PROGRAM MAIN
VAR
  // ── Core robot interface (library FBs) ────────────────────────────────────
  fbStatus     : FB_FanucStatus;        // DI0 byte array → stStatus struct
  fbControl    : FB_FanucControl;       // stControl struct → DO0 byte array
  fbEnable     : FB_FanucEnable;        // Enable sequence state machine
  fbFaultReset : FB_FanucFaultReset;    // Fault reset pulse – FAULT_RESET (UI[5])
  fbStart      : FB_FanucStartProgram;  // Program start (RSR / PNS)
  fbCycleStop  : FB_FanucCycleStop;     // Cycle Stop – CSTOPI (UI[4])
  fbHoming     : FB_FanucHoming;        // Homing sequence – HOME (UI[7])
  stStatus     : ST_FanucStatus;        // Live robot status (inputs)
  stControl    : ST_FanucControl;       // Combined control command (outputs)

  // ── Enable command ────────────────────────────────────────────────────────
  bEnableRobot : BOOL;               // Set TRUE to start enable sequence

  // ── External interlock signals (wire from application safety logic / HMI) ─
  bExtIMSTP  : BOOL;  // Normally Closed: FALSE = software E-stop
  bExtHold   : BOOL;  // Normally Closed: FALSE = pause/hold robot
  bExtSFSPD  : BOOL;  // Normally Closed: FALSE = safe-speed limit active
  bExtStart  : BOOL;  // Start command: forwarded to robot only when in Ready state

  // ── Fault reset ───────────────────────────────────────────────────────────
  bFaultReset  : BOOL;               // Rising edge: send FAULT_RESET pulse (UI[5])

  // ── Cycle Stop ────────────────────────────────────────────────────────────
  bCycleStop   : BOOL;               // Rising edge: send CSTOPI cycle stop command
  eCstopiMode  : E_FanucCstopiMode;  // Must match FANUC "CSTOPI for ABORT" system setting

  // ── Homing ────────────────────────────────────────────────────────────────
  bStartHome   : BOOL;               // Rising edge: start homing sequence (gated by bReady)

  // ── Program start ─────────────────────────────────────────────────────────
  bStartProgram : BOOL;              // Rising edge: start program nProgram (gated by bReady)
  nProgram      : INT := 1;          // Program to start: 1..8 (RSR) or 1..255 (PNS)
  eStartMode    : E_FanucStartMode;  // RSR or PNS – must match FANUC controller UOP config
END_VAR

// 1. Read status – always first
fbStatus(aDI := GVL_Fanuc.DI0, stStatus => stStatus);

// 2. Enable sequence (outputs stControl; other FBs stamp into it below)
fbEnable(
    bEnable   := bEnableRobot,
    stStatus  := stStatus,
    bExtIMSTP := bExtIMSTP,   // Wire from: NOT bSoftEStop
    bExtHold  := bExtHold,    // Wire from: NOT bPauseButton
    bExtSFSPD := bExtSFSPD,   // Wire from: bFenceOK / area scanner
    bExtStart := bExtStart,   // Wire from: HMI start button
    stControl => stControl);

// 3. Program start (VAR_IN_OUT stamps start bits into stControl)
fbStart(
    bStart    := bStartProgram,
    nProgram  := nProgram,
    eMode     := eStartMode,
    bReady    := fbEnable.bReady,
    stStatus  := stStatus,
    stControl := stControl);

// 4. Cycle stop
fbCycleStop(
    bTrigger  := bCycleStop,
    eMode     := eCstopiMode,
    stStatus  := stStatus,
    stControl := stControl);

// 5. Homing
fbHoming(
    bStart    := bStartHome,
    bReady    := fbEnable.bReady,
    stStatus  := stStatus,
    stControl := stControl);

// 6. Fault reset (call when fbEnable.eState = ClearFault and operator requests)
fbFaultReset(
    bReset    := bFaultReset,
    stStatus  := stStatus,
    stControl := stControl);

// 7. Write outputs – always last
fbControl(aDO := GVL_Fanuc.DO0, stControl := stControl);

END_PROGRAM

(* stored: Version 1.1.0.1, ProductVersion 3.1.4026.18
   POU MAIN: Id {6973d23a-8789-7e7c-9fcc-0e3b7f231cb5}, SpecialFunc None *)
